PROGRAM MBUS_HeatCounter_Container (* hier wird die Klemme, an welche der M-Bus mit den Zählern angeschlossen ist, alle 10ms aufgerufen *)
VAR
	Komm_Klemme_WZaehler2		: FB_MBUSKL6781;
	WMZ1						: FB_MBUS_General_Ext;	(*1*)
	WMZ2						: FB_MBUS_General_Ext;	(*1*)

	adrWMZ1			: ST_MBus_SecAdr := (udiIdNumber:=16#13859504);
	adrWMZ2			: ST_MBus_SecAdr := (udiIdNumber:=16#13859500);
	
	fbcatch2 : 	Error_Catch;
END_VAR

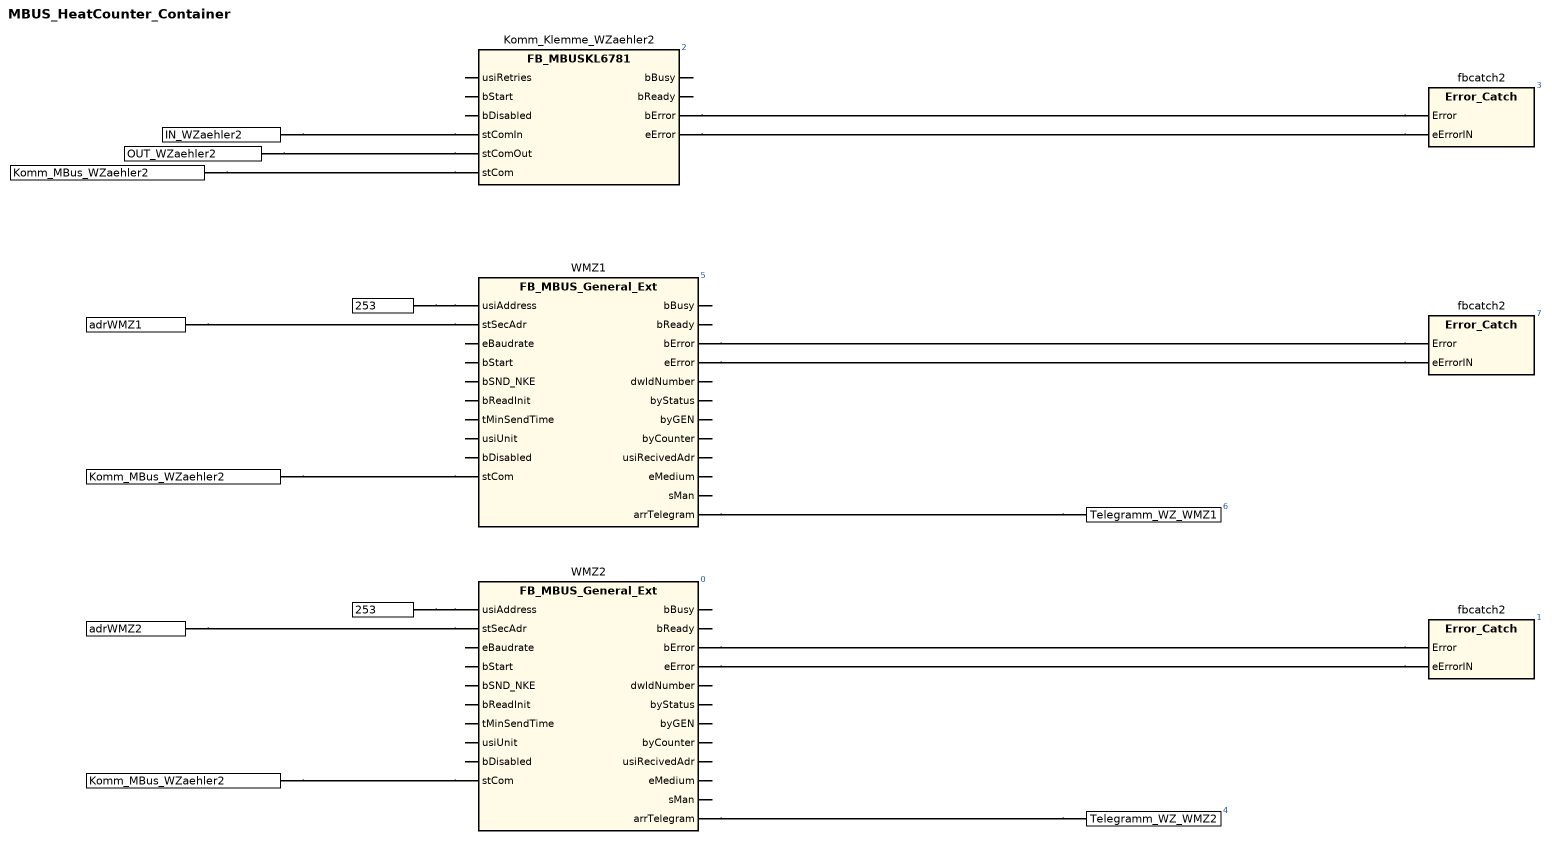
WMZ2(usiAddress := 253, stSecAdr := adrWMZ2, stCom := Komm_MBus_WZaehler2); // FB_MBUS_General_Ext
fbcatch2(Error := WMZ2.bError, eErrorIN := WMZ2.eError); // Error_Catch
Komm_Klemme_WZaehler2(stComIn := IN_WZaehler2, stComOut := OUT_WZaehler2, stCom := Komm_MBus_WZaehler2); // FB_MBUSKL6781
fbcatch2(Error := Komm_Klemme_WZaehler2.bError, eErrorIN := Komm_Klemme_WZaehler2.eError); // Error_Catch
Telegramm_WZ_WMZ2 := WMZ2.arrTelegram;
WMZ1(usiAddress := 253, stSecAdr := adrWMZ1, stCom := Komm_MBus_WZaehler2); // FB_MBUS_General_Ext
Telegramm_WZ_WMZ1 := WMZ1.arrTelegram;
fbcatch2(Error := WMZ1.bError, eErrorIN := WMZ1.eError); // Error_Catch

END_PROGRAM

(* stored: Version 1.1.0.1, ProductVersion 3.1.4024.10
   POU MBUS_HeatCounter_Container: Id {3a3b2554-4e7f-4917-b848-a0dd88abd28f}, SpecialFunc None *)
